FUNCTION SetBit : DWORD
VAR_INPUT
	dPLC_OUT	: DWORD;
	iBitNum		: USINT;
	bstate		: BOOL;
END_VAR
VAR
	bCheckBit	: BOOL;
END_VAR


bCheckBit := DWORD_TO_BOOL(SHR(dPLC_OUT,iBitNum)AND 1);

IF bstate THEN
	dPLC_OUT := SHL(1,iBitNum) OR dPLC_OUT;
ELSE
	IF bCheckbit THEN
		IF dPLC_OUT > 0 THEN
			dPLC_OUT := dPLC_OUT - LREAL_TO_DWORD(EXPT(2,iBitNum));
		END_IF
	END_IF
END_IF

SetBit := dPLC_OUT;

END_FUNCTION

(* stored: Version 1.1.0.1, ProductVersion 3.1.4024.12
   POU SetBit: Id {df8637ce-1772-4c0d-bff2-bb91078cbd62}, SpecialFunc None *)
